			//C6-0x366
			16#366:           //接收C6送来的数据
				//Pre :=BYTE_TO_WORD(frame.data[1]) OR SHL(BYTE_TO_WORD(frame.data[2]),8);
	 			//psYyz^.Status.pressureV8:= 	(Pre-4000)/16000.0*400;	
				//Pre :=BYTE_TO_WORD(frame.data[3]) OR SHL(BYTE_TO_WORD(frame.data[4]),8);
	 			//psYyz^.Status.pressureV9:= 	(Pre-4000)/16000.0*400;	
				pos	:=BYTE_TO_WORD(frame.data[5]) OR SHL(BYTE_TO_WORD(frame.data[6]),8);
				psPVTi^.arrAddtion[1].sPlateStatus.sSensor.Current:=pos*0.1;
				pos	:=BYTE_TO_WORD(frame.data[7]) OR SHL(BYTE_TO_WORD(frame.data[8]),8);
				psPVTi^.arrAddtion[2].sPlateStatus.sSensor.Current:=pos*0.1;
				
		END_CASE
	END_FOR
	gCan.C6RxCounter := gCan.C6RxMsg.RxCounter ;
END_IF

END_FUNCTION

// Device/Application/can/swmc_C12_Rx
FUNCTION swmc_C12_Rx : BOOL
VAR_INPUT
	CNT				: UINT;
	psPVTi			: POINTER TO propValveModule_Ti;
END_VAR
VAR
	frame	 	    : Can_baseframe;
	COB_ID			: UINT;
	I				: UINT;
	Pre				: UINT;
	pos				: WORD;
END_VAR

IF gCan.C12RxMsg.RxCounter <>  gCan.C12RxCounter THEN    //接收到新的数据

	FOR  I := 1 TO  gCan.C12RxMsg.NoOfRxMessages DO
		frame :=CAN_Read_Data_SWMC(12,I);
		COB_ID :=	frame.id;    //获取ID
		CASE COB_ID OF     //根据ID解析协议
		
		
			//C12-0x3C0
			16#3C0:           //接收C12送来的数据
				pos := BYTE_TO_WORD(frame.data[ 1 ]) OR SHL(BYTE_TO_WORD(frame.data[ 2 ]),8);  	
				psPVTi^.arrPV[ 6 ].sNum[ 7 ].posVal.Current:= pos*0.1;	
				pos := BYTE_TO_WORD(frame.data[ 3 ]) OR SHL(BYTE_TO_WORD(frame.data[ 4 ]),8);  
				psPVTi^.arrPV[ 6 ].sNum[ 8 ].posVal.Current:= pos*0.1;		
				pos := BYTE_TO_WORD(frame.data[ 5 ]) OR SHL(BYTE_TO_WORD(frame.data[ 6 ]),8);  
				psPVTi^.arrPV[ 7 ].sNum[ 20 ].posVal.Current:= pos*0.1;	
				pos := BYTE_TO_WORD(frame.data[ 7 ]) OR SHL(BYTE_TO_WORD(frame.data[ 8 ]),8);  	
				psPVTi^.arrPV[ 7 ].sNum[ 21 ].posVal.Current:= pos*0.1;

			//C6-0x3C1
			16#3C1:           //接收C12送来的数据
				pos := BYTE_TO_WORD(frame.data[ 1 ]) OR SHL(BYTE_TO_WORD(frame.data[ 2 ]),8);  	
				psPVTi^.arrPV[ 7 ].sNum[ 1 ].posVal.Current:= pos*0.1;	
				pos := BYTE_TO_WORD(frame.data[ 3 ]) OR SHL(BYTE_TO_WORD(frame.data[ 4 ]),8);  	
				psPVTi^.arrPV[ 7 ].sNum[ 2 ].posVal.Current:= pos*0.1;	
				pos := BYTE_TO_WORD(frame.data[ 5 ]) OR SHL(BYTE_TO_WORD(frame.data[ 6 ]),8);  	
				psPVTi^.arrPV[ 7 ].sNum[ 3 ].posVal.Current:= pos*0.1;	
				pos := BYTE_TO_WORD(frame.data[ 7 ]) OR SHL(BYTE_TO_WORD(frame.data[ 8 ]),8);  	
				psPVTi^.arrPV[ 7 ].sNum[ 4 ].posVal.Current:= pos*0.1;
			//C6-0x3C2
			16#3C2:           //接收C12送来的数据
				pos := BYTE_TO_WORD(frame.data[ 1 ]) OR SHL(BYTE_TO_WORD(frame.data[ 2 ]),8);  	
				psPVTi^.arrPV[ 7 ].sNum[ 5 ].posVal.Current:= pos*0.1;	
				pos := BYTE_TO_WORD(frame.data[ 3 ]) OR SHL(BYTE_TO_WORD(frame.data[ 4 ]),8);  	
				psPVTi^.arrPV[ 7 ].sNum[ 6 ].posVal.Current:= pos*0.1;		
				pos := BYTE_TO_WORD(frame.data[ 5 ]) OR SHL(BYTE_TO_WORD(frame.data[ 6 ]),8);  	
				psPVTi^.arrPV[ 7 ].sNum[ 7 ].posVal.Current:= pos*0.1;		
				pos := BYTE_TO_WORD(frame.data[ 7 ]) OR SHL(BYTE_TO_WORD(frame.data[ 8 ]),8);  	
				psPVTi^.arrPV[ 7 ].sNum[ 8 ].posVal.Current:= pos*0.1;	
			//C6-0x3C3
			16#3C3:           //接收C12送来的数据
				pos := BYTE_TO_WORD(frame.data[ 1 ]) OR SHL(BYTE_TO_WORD(frame.data[ 2 ]),8);  	
				psPVTi^.arrPV[ 7 ].sNum[ 9 ].posVal.Current:= pos*0.1;		
				pos := BYTE_TO_WORD(frame.data[ 3 ]) OR SHL(BYTE_TO_WORD(frame.data[ 4 ]),8);  	
				psPVTi^.arrPV[ 7 ].sNum[ 22 ].posVal.Current:= pos*0.1;		
				pos := BYTE_TO_WORD(frame.data[ 5 ]) OR SHL(BYTE_TO_WORD(frame.data[ 6 ]),8);  	
				psPVTi^.arrPV[7 ].sNum[ 23 ].posVal.Current:= pos*0.1;		
				pos := BYTE_TO_WORD(frame.data[ 7 ]) OR SHL(BYTE_TO_WORD(frame.data[ 8 ]),8);  	
				psPVTi^.arrPV[ 1 ].sNum[ 1 ].posVal.Current:= pos*0.1;	
			//C6-0x3C4
			16#3C4:           //接收C12送来的数据
				pos := BYTE_TO_WORD(frame.data[ 1 ]) OR SHL(BYTE_TO_WORD(frame.data[ 2 ]),8);  	
				psPVTi^.arrPV[ 1 ].sNum[ 2 ].posVal.Current:= pos*0.1;		
				pos := BYTE_TO_WORD(frame.data[ 3 ]) OR SHL(BYTE_TO_WORD(frame.data[ 4 ]),8);  	
				psPVTi^.arrPV[ 7 ].sNum[ 10 ].posVal.Current:= pos*0.1;		
				pos := BYTE_TO_WORD(frame.data[ 5 ]) OR SHL(BYTE_TO_WORD(frame.data[ 6 ]),8);  	
				psPVTi^.arrPV[ 7 ].sNum[ 11 ].posVal.Current:= pos*0.1;		
				pos := BYTE_TO_WORD(frame.data[ 7 ]) OR SHL(BYTE_TO_WORD(frame.data[ 8 ]),8);  	
				psPVTi^.arrPV[7 ].sNum[ 12 ].posVal.Current:= pos*0.1;	
			//C6-0x3C5
			16#3C5:           //接收C12送来的数据
				pos := BYTE_TO_WORD(frame.data[ 1 ]) OR SHL(BYTE_TO_WORD(frame.data[ 2 ]),8);  	
				psPVTi^.arrPV[ 7 ].sNum[ 13 ].posVal.Current:= pos*0.1;		
				pos := BYTE_TO_WORD(frame.data[ 3 ]) OR SHL(BYTE_TO_WORD(frame.data[ 4 ]),8);  	
				psPVTi^.arrPV[ 7 ].sNum[ 14 ].posVal.Current:= pos*0.1;		
				pos := BYTE_TO_WORD(frame.data[ 5 ]) OR SHL(BYTE_TO_WORD(frame.data[ 6 ]),8);  	
				psPVTi^.arrPV[ 7 ].sNum[ 15 ].posVal.Current:= pos*0.1;		
				pos := BYTE_TO_WORD(frame.data[ 7 ]) OR SHL(BYTE_TO_WORD(frame.data[ 8 ]),8);  	
				psPVTi^.arrPV[ 7 ].sNum[ 16 ].posVal.Current:= pos*0.1;
			//C6-0x3C6
			16#3C6:           //接收C12送来的数据
				pos := BYTE_TO_WORD(frame.data[ 1 ]) OR SHL(BYTE_TO_WORD(frame.data[ 2 ]),8);  	
				psPVTi^.arrPV[ 7 ].sNum[ 17 ].posVal.Current:= pos*0.1;		
				pos := BYTE_TO_WORD(frame.data[ 3 ]) OR SHL(BYTE_TO_WORD(frame.data[ 4 ]),8);  	
				psPVTi^.arrPV[ 7 ].sNum[ 18 ].posVal.Current:= pos*0.1;		
				pos := BYTE_TO_WORD(frame.data[ 5 ]) OR SHL(BYTE_TO_WORD(frame.data[ 6 ]),8);  	
				psPVTi^.arrPV[ 7 ].sNum[ 19 ].posVal.Current:= pos*0.1;		
						
		
			
		END_CASE
	END_FOR
	gCan.C12RxCounter := gCan.C12RxMsg.RxCounter ;
END_IF

END_FUNCTION

// Device/Application/dataUpload/fileSaver
PROGRAM fileSaver
VAR
	path 			:STRING:='D:/log';
	intervalMs		:INT := 10;		//间隔时间
	
	init			:BOOL:= TRUE;
	i0				:INT;
	i1				:INT;	
	cCtrl			:INT;

	sav				:ARRAY[1..7,1..24] OF fileSave;
	getCtrl			:findMasterCtrl;
	getStat			:getStateByIdx;
	speed			:INT;
	nowCmd			:ARRAY[1..7,1..24] OF BOOL;
	canWrite		:ARRAY[1..7,1..24] OF BOOL;
	nowPosition		:ARRAY[1..7,1..24] OF INT;
	lastPosition	:ARRAY[1..7,1..24] OF INT;
	state			:ARRAY[1..7,1..24] OF INT;
	flag			:ARRAY[1..7,1..24] OF INT;
END_VAR
VAR CONSTANT
	aOil	:ARRAY [1..7] OF INT :=[9,11,8,8,8,8,23];		
END_VAR


//initialize
IF init THEN
	init := FALSE;
	FOR i0:=1 TO 7 DO	
	FOR i1:=1 TO aOil[i0] DO	
		sav[i0,i1](filePath := path, intervalt := intervalMs);
		sav[i0,i1].createDir(gUI.TiG_NameInit.strName[i0,i1]);
	END_FOR	
	END_FOR	
END_IF

//detect and record
FOR i0:=1 TO 7 DO		
	FOR i1:=1 TO aOil[i0] DO
		//get command
		getCtrl(grp := i0, num := i1, ctrl => cCtrl);
		nowCmd[i0,i1] := gUI.TiG.arrPV[i0].sColumn[cCtrl].bExtend OR gUI.TiG.arrPV[i0].sColumn[cCtrl].bRetract;
		//device is running
		IF nowCmd[i0 ,i1] THEN
			IF flag[i0,i1] = 0 THEN
				sav[i0,i1].new(devName :=gUI.TiG_NameInit.strName[i0,i1]);
				flag[i0,i1] := 1;
			END_IF
			//prepare data
			getData();
			//write
			sav[i0,i1].write(positionInt:=nowPosition[i0,i1],speedInt:= speed,
				stateInt := state[i0,i1]);
			
		ELSE
			//stop recording when command ends
			IF flag[i0,i1] = 1 THEN
				sav[i0,i1].write(positionInt:=nowPosition[i0,i1],speedInt:= speed,
								stateInt := state[i0,i1]);
				sav[i0,i1].close();
				flag[i0,i1] := 0;
			END_IF
		END_IF
	END_FOR	
END_FOR

ACTION getData:

//进制转换 到0.01mm
lastPosition[i0, i1] := nowPosition[i0, i1];
nowPosition[i0, i1] := REAL_TO_INT(10 * gImple.PV_GroupTi.arrPV[i0].sNum[i1].posVal.Current);

//speed  -  mm/s
IF nowPosition[i0, i1] > lastPosition[i0, i1] THEN
	speed := (nowPosition[i0, i1] - lastPosition[i0, i1]) * 100 / intervalMs;
ELSE
	speed := (lastPosition[i0, i1] - nowPosition[i0, i1]) * 100 / intervalMs;
END_IF

getStat(grp := i0, ctrl := cCtrl,state => state[i0, i1]);
END_ACTION

END_PROGRAM

// Device/Application/dataUpload/fileSave
FUNCTION_BLOCK fileSave
VAR_INPUT
	filePath 	:STRING;
	intervalt	:INT;
END_VAR
VAR_OUTPUT
END_VAR
VAR
	
	lineCount	: INT;
	fileHandle  : DWORD;
	fileName	: STRING;
END_VAR

METHOD new

	
VAR_INPUT
	devName		: STRING ;

END_VAR
VAR
	
	fileHandle0 : DWORD;
	datetime	: DATE_AND_TIME;
	UdIntms 	: UDINT;
	UdMsOffset  : UDINT;
	DTimer_Str  : STRING;
	uiYear 		: UINT; 
    uiMonth 	: UINT; 
    uiDay 		: UINT; 
    uiHour 		: UINT; 
    uiMinute 	: UINT; 
    uiSecond 	: UINT;	
	uiMsSecond	: UINT;



	 S_Time64		:  SysTime64;
	 STT			:  CurTimeEx;
	 S_Time			:  SystemTimeDate;
	 Time_Str		:  STRING;
	F_err		: DWORD;
	F_HANDL		: DWORD;

END_VAR

	STT(SystemTime:= S_Time64, TimeDate:= S_Time);
	Time_Str :='';
	Time_Str := concat(Time_Str,UINT_TO_STRING(S_Time.Year));
	Time_Str := concat(Time_Str,'-');
	Time_Str := concat(Time_Str,UINT_TO_STRING(S_Time.Month));
	Time_Str := concat(Time_Str,'-');
	Time_Str := concat(Time_Str,UINT_TO_STRING(S_Time.Day));
	Time_Str := concat(Time_Str,'_');
	Time_Str := concat(Time_Str,UINT_TO_STRING(S_Time.Hour));
	Time_Str := concat(Time_Str,'-');
	Time_Str := concat(Time_Str,UINT_TO_STRING(S_Time.Minute));
	Time_Str := concat(Time_Str,'-');
	Time_Str := concat(Time_Str,UINT_TO_STRING(S_Time.Second));
	Time_Str := concat(Time_Str,'_');
	Time_Str := concat(Time_Str,UINT_TO_STRING(S_Time.Milliseconds));

	fileName := FilePath;
	fileName := concat(fileName,'/');
	fileName := concat(fileName,devName);

	
	fileName := concat(fileName,'/');
	fileName := concat(fileName,devName);
	fileName := concat(fileName,'-');
	fileName := concat(fileName,Time_Str);
    fileName := concat(fileName,'.txt');

	fileHandle := SysFileOpen(szFile:= fileName, am:=ACCESS_MODE.AM_WRITE, pResult:= ADR(F_err));
	lineCount := -1;
	//fileHandle := SysFileOpen(szFile:= fileName, am:=ACCESS_MODE.AM_APPEND, pResult:= ADR(F_err));
END_METHOD

METHOD close
VAR_INPUT
END_VAR
IF fileHandle <> 0 THEN
	SysFileClose(hFile := fileHandle);
	fileHandle := 0;
END_IF
END_METHOD

METHOD write
VAR_INPUT

	positionInt 	:INT;
	speedInt 		:INT;
	stateInt		:INT;
	
END_VAR
VAR
	data		: STRING;
	F_err		: DWORD;
	tempInt		: INT;
END_VAR

IF fileHandle <> 0 THEN
	lineCount := lineCount + 1;
	tempInt	:= lineCount * intervalt;
	data := INT_TO_STRING(lineCount);
	data := concat(data,'$T$T');
	data := concat(data, INT_TO_STRING(tempInt));
	IF tempInt < 1000 THEN
		data := concat(data,'$T');
	END_IF
	data := concat(data,'$T$T');
	data := concat(data,INT_TO_STRING(positionInt));
	data := concat(data,'$T');
	data := concat(data,INT_TO_STRING(speedInt));
	data := concat(data,'$T');
	data := concat(data,INT_TO_STRING(stateInt));
	data := concat(data,'$R');
	
	SysFileWrite(hFile:=fileHandle , pbyBuffer:= ADR(data) , ulSize:= SysStrLen(data) , pResult:= ADR(F_err));		// 写入数据

END_IF
END_METHOD

METHOD createDir
VAR_INPUT
	devName		: STRING ;
END_VAR
VAR
	filePath1	:STRING;
END_VAR
filePath1 := FilePath;
filePath1 := concat(filePath1,'/');
filePath1 := concat(filePath1,devName);
SysDirCreate2(filePath1, TRUE);
END_METHOD

END_FUNCTION_BLOCK

// Device/Application/public_datum/datarecord/datSave
FUNCTION_BLOCK datSave
VAR_INPUT
	Data_Arry	: ARRAY[1..200] OF UINT;	// 数据输入 一次最大可以写入200个数据
	Num			: UINT;						// 存储数据个数
	FilePath 	: STRING := 'C:/DataSave'; 	// 存储文件夹
	cycle		: TIME;						// 更新一个文件夹时间
END_VAR
VAR_OUTPUT
END_VAR
VAR
	datetime	: DATE_AND_TIME;
	uiYear 		: UINT; 
    uiMonth 	: UINT; 
    uiDay 		: UINT; 
    uiHour 		: UINT; 
    uiMinute 	: UINT; 
    uiSecond 	: UINT;	
	uiMsSecond	: UINT;
	Last_S		: UINT:=100;
	UdMsOffset  : UDINT;
	UdIntms 	: UDINT;
	DTimer_Arry : ARRAY[1..7] OF UINT;
END_VAR
VAR
	File_Init	: BOOL :=TRUE;
	Frame_Cnt	: LINT;
	Data_Save_Init :BOOL:=TRUE;
	New_File_Ton: TON;
	Filename	: STRING;
	F_HANDL		: DWORD;
	F_err		: DWORD;
	F_pos		: DWORD;
END_VAR

datetime:=GetDateTime();   //获取时间
DTU.DTSplit(
		dtDateAndTime:= datetime, 
		puiYear:= ADR(uiYear), 
		puiMonth:=  ADR(uiMonth), 
		puiDay:=  ADR(uiDay), 
		puiHour:=  ADR(uiHour), 
		puiMinute:=  ADR(uiMinute), 
		puiSecond:= ADR(uiSecond) );

IF  Data_Save_Init THEN			//数据存储初始化
	IF uiSecond = Last_S +1 OR  uiSecond = Last_S -59 THEN
		UdMsOffset := SysTimeGetMs();
		Last_S :=  uiSecond;
	ELSE
		Last_S :=  uiSecond;
		RETURN;
	END_IF
    Data_Save_Init := FALSE;
END_IF

IF 	File_Init  THEN          //创建文件
	Filename := FilePath;
	Filename := concat(Filename,'/');
	Filename := concat(Filename,UINT_TO_STRING(uiYear));
	Filename := concat(Filename,'_');
	Filename := concat(Filename,UINT_TO_STRING(uiMonth));
	Filename := concat(Filename,'_');
	Filename := concat(Filename,UINT_TO_STRING(uiDay));
	Filename := concat(Filename,'_');
	Filename := concat(Filename,UINT_TO_STRING(uiHour+8));
 	Filename := concat(Filename,'_');
	Filename := concat(Filename,UINT_TO_STRING(uiMinute));
	Filename := concat(Filename,'_');
	Filename := concat(Filename,UINT_TO_STRING(uiSecond));
    Filename := concat(Filename,'_Data.bin');
	Frame_Cnt := 0;
	F_HANDL :=SysFileOpen(szFile:= Filename, am:=ACCESS_MODE.AM_WRITE, pResult:= ADR(F_err));  //创建新文件
	SysFileClose(hFile:=F_HANDL );
	File_Init := FALSE;
	New_File_Ton(IN:= FALSE , PT:= cycle, Q=> , ET=> );  //复位
END_IF

New_File_Ton(IN:= TRUE , PT:= cycle, Q=> , ET=> );			//4小时创建一个新文件
IF New_File_Ton.Q THEN
	File_Init := TRUE;	
END_IF



UdIntms := SysTimeGetMs();
DTimer_Arry[1] := uiYear;
DTimer_Arry[2] := uiMonth;
DTimer_Arry[3] := uiDay;
DTimer_Arry[4] := uiHour+8;
DTimer_Arry[5] := uiMinute;
DTimer_Arry[6] := uiSecond;
DTimer_Arry[7] := UDINT_TO_UINT((UdIntms - UdMsOffset)MOD 1000);

Frame_Cnt := Frame_Cnt + 1;    	//帧计数增加

F_HANDL :=SysFileOpen(szFile:= Filename, am:=ACCESS_MODE.AM_APPEND, pResult:= ADR(F_err));  //打开文件
SysFileGetPos(hFile:= F_HANDL , pulPos:= ADR(F_pos));		//获取文件位置
SysFileSetPos(hFile:= F_HANDL, ulOffset:= 0);	//设置帧位置
SysFileWrite(hFile:=F_HANDL , pbyBuffer:= ADR(Frame_Cnt) , ulSize:= SIZEOF(Frame_Cnt) , pResult:= ADR(F_err));    //修改总帧数
IF F_pos <> 0 THEN		//不是新文件，设置写入位置
	SysFileSetPos(hFile:= F_HANDL, ulOffset:= F_pos);
END_IF
SysFileWrite(hFile:=F_HANDL , pbyBuffer:= ADR(DTimer_Arry) , ulSize:= SIZEOF(DTimer_Arry) , pResult:= ADR(F_err));  // 保存时间
SysFileWrite(hFile:=F_HANDL , pbyBuffer:= ADR(Data_Arry) , ulSize:= SIZEOF(UINT)*Num , pResult:= ADR(F_err));		// 保存数据
SysFileClose(hFile:=F_HANDL );

END_FUNCTION_BLOCK

// Device/Application/rail_ceiling/positionRecord
PROGRAM positionRecord
VAR
	arrPosVal			:ARRAY[1..200] OF UINT;
	fbDatSav			:DatSave;
	iT1					:UINT;
	iT2					:UINT;
	iNum				:UINT;
END_VAR
VAR CONSTANT
	aOil	:ARRAY [1..7] OF UINT :=[9,11,8,8,8,8,23];		
END_VAR

iNum:=1;
FOR iT1:=1 TO 7 DO
	FOR iT2:=1 TO aOil[iT1] DO
		arrPosVal[iNum]:=REAL_TO_UINT(gImple.PV_GroupTi.arrPV[iT1].sNum[iT2].posVal.Current);
		iNum:=iNum+1;
	END_FOR
END_FOR
fbDatSav(Data_Arry:=arrPosVal , Num:= 75 , FilePath:= 'D:/DataSave', cycle:= T#7200S);

END_PROGRAM

// Device/Application/public_datum/cmdcheck/syncUnitCheck
FUNCTION_BLOCK syncUnitCheck
VAR_INPUT
	arrPosVal	:ARRAY  [1..2] OF OilBlockUnit_Status_PosVal;

	cmdAct		:cmdStat;
	
END_VAR
VAR_OUTPUT
	bFetch		:BOOL;
END_VAR
VAR
	iCheck			:INT;
	iNum			:INT;				//有值的位移传感器值
	outStat			:ARRAY[1..2] OF OilBlockUnit_Status_Loc;
	iTemp			:INT;
	bAllDone		:BOOL;
END_VAR

iNum:=0;
FOR iTemp :=1 TO 2 DO
	IF arrPosVal[iTemp].Extend <> 0 THEN
		iNum:=iNum+1;
	END_IF
END_FOR
FOR iCheck:=1 TO iNum DO
	outStat[iCheck]	:=fGetUnitStat(arrPosVal[iCheck].Extend,arrPosVal[iCheck].Retract,arrPosVal[iCheck].Current,2.0);
END_FOR


bAllDone:=TRUE;

	//有一个未到指令位置则未完成
	CASE cmdAct OF 
		cmdStat.cExtend:
			FOR iCheck:=1 TO iNum DO
				IF outStat[iCheck]<>OilBlockUnit_Status_Loc.eExtended THEN
					bAllDone:=FALSE;
				END_IF
			END_FOR
		cmdStat.cRetract:
			FOR iCheck:=1 TO iNum DO
				IF outStat[iCheck]<>OilBlockUnit_Status_Loc.eRetracted THEN
					bAllDone:=FALSE;
				END_IF
			END_FOR	
		cmdStat.cStop:
			
	END_CASE

IF bAllDone THEN
	bFetch	:= TRUE;
ELSE
	bFetch	:= FALSE;
END_IF

END_FUNCTION_BLOCK

// Device/Application/display/Module/OilBlock_PrimButton
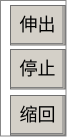
VISUALIZATION OilBlock_PrimButton  // 67x137
VAR_IN_OUT
	extendButton		: BOOL;
	retractButton		: BOOL;
	stopButton			: BOOL;
	
END_VAR
    Button (10,95 55x40), "缩回"
        toggle retractButton
    Button (10,49 55x40), "停止"
        toggle stopButton
    Button (10,5 55x40), "伸出"
        toggle extendButton
END_VISUALIZATION

// Device/Application/display/Module/OilBlock_PrimInfo
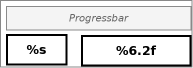
VISUALIZATION OilBlock_PrimInfo  // 193x68
VAR_IN_OUT
	nameStr		:STRING;
	posVal		:REAL;
	percentBar	:REAL;
END_VAR
    RoundedRectangle (6,34 61x31), "%s", text variable: nameStr
    RoundedRectangle (81,35 110x31), "%6.2f", text variable: posVal
    Progressbar (6,6 185x24), variable: percentBar
END_VISUALIZATION

// Device/Application/display/Module/ModuleX2
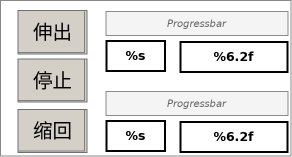
VISUALIZATION ModuleX2  // 292x157
VAR_IN_OUT
	extendButton		: BOOL;
	retractButton		: BOOL;
	stopButton			: BOOL;
	
	nameStr1			:STRING;
	posVal1				:REAL;
	percentBar1			:REAL;
	nameStr2			:STRING;
	posVal2				:REAL;
	percentBar2			:REAL;
END_VAR
    Group (5,5 285x150)
        Frame (0,0 85x150)
            shows OilBlock_PrimButton(extendButton := extendButton, retractButton := retractButton, stopButton := stopButton)
        Frame (95,0 190x70)
            shows OilBlock_PrimInfo(nameStr := nameStr1, posVal := posVal1, percentBar := percentBar1)
        Frame (95,80 190x70)
            shows OilBlock_PrimInfo(nameStr := nameStr2, posVal := posVal2, percentBar := percentBar2)
END_VISUALIZATION

// Device/Application/display/Module/ModuleX1
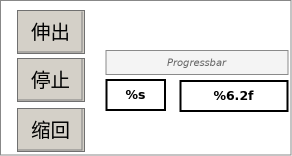
VISUALIZATION ModuleX1  // 292x156
VAR_IN_OUT
	extendButton		: BOOL;
	retractButton		: BOOL;
	stopButton			: BOOL;
	
	nameStr				:STRING;
	posVal				:REAL;
	percentBar			:REAL;
END_VAR
    Group (5,5 285x149)
        Frame (0,0 82x149)
            shows OilBlock_PrimButton(extendButton := extendButton, retractButton := retractButton, stopButton := stopButton)
        Frame (95,39 190x70)
            shows OilBlock_PrimInfo(nameStr := nameStr, posVal := posVal, percentBar := percentBar)
END_VISUALIZATION

// Device/Application/display/Module/ModuleX3
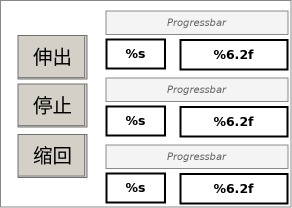
VISUALIZATION ModuleX3  // 292x208
VAR_IN_OUT
	extendButton		: BOOL;
	retractButton		: BOOL;
	stopButton			: BOOL;
	
	nameStr1			:STRING;
	posVal1				:REAL;
	percentBar1			:REAL;
	nameStr2			:STRING;
	posVal2				:REAL;
	percentBar2			:REAL;
	nameStr3			:STRING;
	posVal3				:REAL;
	percentBar3			:REAL;
END_VAR
    Group (5,5 285x201)
        Frame (0,25 85x150)
            shows OilBlock_PrimButton(extendButton := extendButton, retractButton := retractButton, stopButton := stopButton)
        Frame (95,0 190x67)
            shows OilBlock_PrimInfo(nameStr := nameStr1, posVal := posVal1, percentBar := percentBar1)
        Frame (95,67 190x67)
            shows OilBlock_PrimInfo(nameStr := nameStr2, posVal := posVal2, percentBar := percentBar2)
        Frame (95,134 190x67)
            shows OilBlock_PrimInfo(nameStr := nameStr3, posVal := posVal3, percentBar := percentBar3)
END_VISUALIZATION

// Device/Application/display/Module/ModuleX8
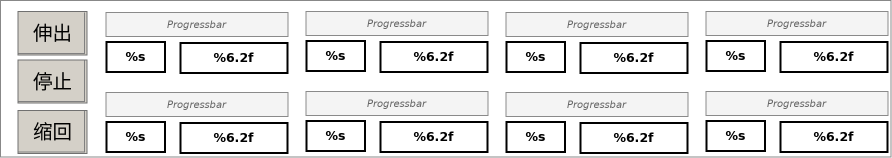
VISUALIZATION ModuleX8  // 892x158
VAR_IN_OUT
	extendButton		: BOOL;
	retractButton		: BOOL;
	stopButton			: BOOL;
	
	nameStr1			:STRING;
	posVal1				:REAL;
	percentBar1			:REAL;
	
	nameStr2			:STRING;
	posVal2				:REAL;
	percentBar2			:REAL;
	
	nameStr3			:STRING;
	posVal3				:REAL;
	percentBar3			:REAL;
	
	nameStr4			:STRING;
	posVal4				:REAL;
	percentBar4			:REAL;
	
	nameStr5			:STRING;
	posVal5				:REAL;
	percentBar5			:REAL;
	
	nameStr6			:STRING;
	posVal6				:REAL;
	percentBar6			:REAL;
	
	nameStr7			:STRING;
	posVal7				:REAL;
	percentBar7			:REAL;
	
	nameStr8			:STRING;
	posVal8				:REAL;
	percentBar8			:REAL;	
	
END_VAR
    Group (5,5 885x151)
        Frame (0,1 85x150)
            shows OilBlock_PrimButton(extendButton := extendButton, retractButton := retractButton, stopButton := stopButton)
        Group (95,0 390x151)
            Group (0,1 190x150)
                Frame (0,0 190x70)
                    shows OilBlock_PrimInfo(nameStr := nameStr1, posVal := posVal1, percentBar := percentBar1)
                Frame (0,80 190x70)
                    shows OilBlock_PrimInfo(nameStr := nameStr2, posVal := posVal2, percentBar := percentBar2)
            Frame (200,0 190x70)
                shows OilBlock_PrimInfo(nameStr := nameStr3, posVal := posVal3, percentBar := percentBar3)
            Frame (200,80 190x70)
                shows OilBlock_PrimInfo(nameStr := nameStr4, posVal := posVal4, percentBar := percentBar4)
        Frame (495,1 190x70)
            shows OilBlock_PrimInfo(nameStr := nameStr5, posVal := posVal5, percentBar := percentBar5)
        Frame (495,81 190x70)
            shows OilBlock_PrimInfo(nameStr := nameStr6, posVal := posVal6, percentBar := percentBar6)
        Frame (695,0 190x70)
            shows OilBlock_PrimInfo(nameStr := nameStr7, posVal := posVal7, percentBar := percentBar7)
        Frame (695,80 190x70)
            shows OilBlock_PrimInfo(nameStr := nameStr8, posVal := posVal8, percentBar := percentBar8)
END_VISUALIZATION

// Device/Application/display/Module/ModuleX4
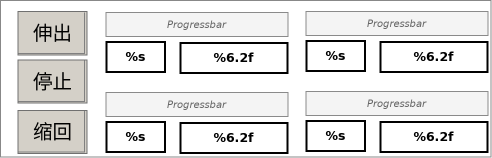
VISUALIZATION ModuleX4  // 492x158
VAR_IN_OUT
	extendButton		: BOOL;
	retractButton		: BOOL;
	stopButton			: BOOL;
	
	nameStr1			:STRING;
	posVal1				:REAL;
	percentBar1			:REAL;
	nameStr2			:STRING;
	posVal2				:REAL;
	percentBar2			:REAL;
	nameStr3			:STRING;
	posVal3				:REAL;
	percentBar3			:REAL;
	nameStr4			:STRING;
	posVal4				:REAL;
	percentBar4			:REAL;
	
	
END_VAR
    Group (5,5 485x151)
        Frame (0,1 85x150)
            shows OilBlock_PrimButton(extendButton := extendButton, retractButton := retractButton, stopButton := stopButton)
        Group (95,1 190x150)
            Frame (0,0 190x70)
                shows OilBlock_PrimInfo(nameStr := nameStr1, posVal := posVal1, percentBar := percentBar1)
            Frame (0,80 190x70)
                shows OilBlock_PrimInfo(nameStr := nameStr2, posVal := posVal2, percentBar := percentBar2)
        Frame (295,0 190x70)
            shows OilBlock_PrimInfo(nameStr := nameStr3, posVal := posVal3, percentBar := percentBar3)
        Frame (295,80 190x70)
            shows OilBlock_PrimInfo(nameStr := nameStr4, posVal := posVal4, percentBar := percentBar4)
END_VISUALIZATION

// Device/Application/display/Module/ModuleX5
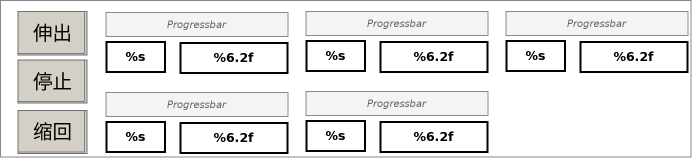
VISUALIZATION ModuleX5  // 692x158
VAR_IN_OUT
	extendButton		: BOOL;
	retractButton		: BOOL;
	stopButton			: BOOL;
	
	nameStr1			:STRING;
	posVal1				:REAL;
	percentBar1			:REAL;
	nameStr2			:STRING;
	posVal2				:REAL;
	percentBar2			:REAL;
	nameStr3			:STRING;
	posVal3				:REAL;
	percentBar3			:REAL;
	nameStr4			:STRING;
	posVal4				:REAL;
	percentBar4			:REAL;
	nameStr5			:STRING;
	posVal5				:REAL;
	percentBar5			:REAL;
	
	
END_VAR
    Group (5,5 685x151)
        Frame (0,1 85x150)
            shows OilBlock_PrimButton(extendButton := extendButton, retractButton := retractButton, stopButton := stopButton)
        Group (95,1 190x150)
            Frame (0,0 190x70)
                shows OilBlock_PrimInfo(nameStr := nameStr1, posVal := posVal1, percentBar := percentBar1)
            Frame (0,80 190x70)
                shows OilBlock_PrimInfo(nameStr := nameStr2, posVal := posVal2, percentBar := percentBar2)
        Frame (295,0 190x70)
            shows OilBlock_PrimInfo(nameStr := nameStr3, posVal := posVal3, percentBar := percentBar3)
        Frame (295,80 190x70)
            shows OilBlock_PrimInfo(nameStr := nameStr4, posVal := posVal4, percentBar := percentBar4)
        Frame (495,0 190x70)
            shows OilBlock_PrimInfo(nameStr := nameStr5, posVal := posVal5, percentBar := percentBar5)
END_VISUALIZATION

// Device/Application/display/OrigTi/Ceiling_Rail2
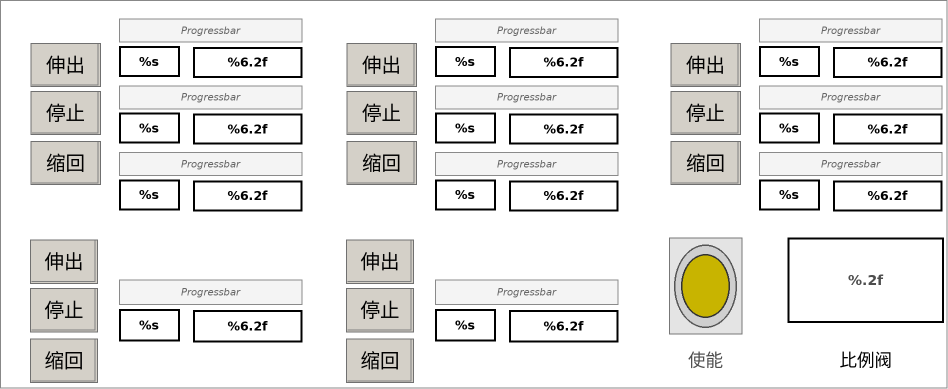
VISUALIZATION Ceiling_Rail2  // 948x389
    Frame (13,8 293x207)
        shows ModuleX3(extendButton := gUI.TiG.arrPV[2].sColumn[1].bExtend, retractButton := gUI.TiG.arrPV[2].sColumn[1].bRetract, stopButton := gUI.TiG.arrPV[2].sColumn[1].bStop, nameStr1 := gUI.TiG.arrPV[2].sNum[1].strName, posVal1 := gUI.TiG.arrPV[2].sNum[1].rPosition, percentBar1 := gUI.TiG.arrPV[2].sNum[1].rPercent, nameStr2 := gUI.TiG.arrPV[2].sNum[2].strName, posVal2 := gUI.TiG.arrPV[2].sNum[2].rPosition, percentBar2 := gUI.TiG.arrPV[2].sNum[2].rPercent, nameStr3 := gUI.TiG.arrPV[2].sNum[3].strName, posVal3 := gUI.TiG.arrPV[2].sNum[3].rPosition, percentBar3 := gUI.TiG.arrPV[2].sNum[3].rPercent)
    Frame (13,229 293x158)
        shows ModuleX1(extendButton := gUI.TiG.arrPV[2].sColumn[2].bExtend, retractButton := gUI.TiG.arrPV[2].sColumn[2].bRetract, stopButton := gUI.TiG.arrPV[2].sColumn[2].bStop, nameStr := gUI.TiG.arrPV[2].sNum[4].strName, posVal := gUI.TiG.arrPV[2].sNum[4].rPosition, percentBar := gUI.TiG.arrPV[2].sNum[4].rPercent)
    Frame (329,8 293x207)
        shows ModuleX3(extendButton := gUI.TiG.arrPV[2].sColumn[3].bExtend, retractButton := gUI.TiG.arrPV[2].sColumn[3].bRetract, stopButton := gUI.TiG.arrPV[2].sColumn[3].bStop, nameStr1 := gUI.TiG.arrPV[2].sNum[5].strName, posVal1 := gUI.TiG.arrPV[2].sNum[5].rPosition, percentBar1 := gUI.TiG.arrPV[2].sNum[5].rPercent, nameStr2 := gUI.TiG.arrPV[2].sNum[6].strName, posVal2 := gUI.TiG.arrPV[2].sNum[6].rPosition, percentBar2 := gUI.TiG.arrPV[2].sNum[6].rPercent, nameStr3 := gUI.TiG.arrPV[2].sNum[7].strName, posVal3 := gUI.TiG.arrPV[2].sNum[7].rPosition, percentBar3 := gUI.TiG.arrPV[2].sNum[7].rPercent)
    Frame (329,229 293x158)
        shows ModuleX1(extendButton := gUI.TiG.arrPV[2].sColumn[4].bExtend, retractButton := gUI.TiG.arrPV[2].sColumn[4].bRetract, stopButton := gUI.TiG.arrPV[2].sColumn[4].bStop, nameStr := gUI.TiG.arrPV[2].sNum[8].strName, posVal := gUI.TiG.arrPV[2].sNum[8].rPosition, percentBar := gUI.TiG.arrPV[2].sNum[8].rPercent)
    Frame (653,8 293x207)
        shows ModuleX3(extendButton := gUI.TiG.arrPV[2].sColumn[5].bExtend, retractButton := gUI.TiG.arrPV[2].sColumn[5].bRetract, stopButton := gUI.TiG.arrPV[2].sColumn[5].bStop, nameStr1 := gUI.TiG.arrPV[2].sNum[9].strName, posVal1 := gUI.TiG.arrPV[2].sNum[9].rPosition, percentBar1 := gUI.TiG.arrPV[2].sNum[9].rPercent, nameStr2 := gUI.TiG.arrPV[2].sNum[10].strName, posVal2 := gUI.TiG.arrPV[2].sNum[10].rPosition, percentBar2 := gUI.TiG.arrPV[2].sNum[10].rPercent, nameStr3 := gUI.TiG.arrPV[2].sNum[11].strName, posVal3 := gUI.TiG.arrPV[2].sNum[11].rPosition, percentBar3 := gUI.TiG.arrPV[2].sNum[11].rPercent)
    Frame (653,229 293x158)
        shows ModuleDTD(enable := gUI.TiG.arrPV[2].bPVD_enable, propPercent := gUI.TiG.arrPV[2].rPVDPercent)
END_VISUALIZATION

// Device/Application/display/Module/ModuleDTD
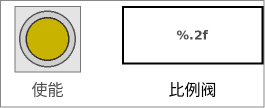
VISUALIZATION ModuleDTD  // 265x108
VAR_IN_OUT
	enable			:BOOL;
	propPercent		:REAL;
END_VAR
    Rectangle (122,6 141x58), "%.2f", text variable: propPercent
        OnMouseDown: write the text variable via Default, min 0, max 100
    Label (122,74 141x32), "比例阀"
    PushSwitchLed (13,6 69x66), variable: enable, behaviour: TOGGLE, style: Switch-PushSwitchLed-Yellow
    Label (13,74 69x32), "使能"
END_VISUALIZATION

// Device/Application/display/OrigTi/Ceiling_Rail1
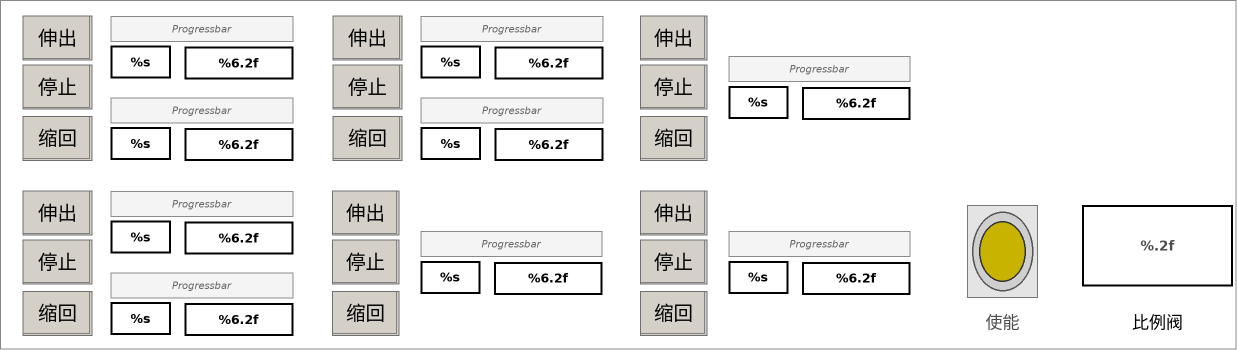
VISUALIZATION Ceiling_Rail1  // 1237x350
    Frame (5,5 292x160)
        shows ModuleX2(extendButton := gUI.TiG.arrPV[1].sColumn[1].bExtend, retractButton := gUI.TiG.arrPV[1].sColumn[1].bRetract, stopButton := gUI.TiG.arrPV[1].sColumn[1].bStop, nameStr1 := gUI.TiG.arrPV[1].sNum[1].strName, posVal1 := gUI.TiG.arrPV[1].sNum[1].rPosition, percentBar1 := gUI.TiG.arrPV[1].sNum[1].rPercent, nameStr2 := gUI.TiG.arrPV[1].sNum[2].strName, posVal2 := gUI.TiG.arrPV[1].sNum[2].rPosition, percentBar2 := gUI.TiG.arrPV[1].sNum[2].rPercent)
    Frame (315,5 292x160)
        shows ModuleX2(extendButton := gUI.TiG.arrPV[1].sColumn[2].bExtend, retractButton := gUI.TiG.arrPV[1].sColumn[2].bRetract, stopButton := gUI.TiG.arrPV[1].sColumn[2].bStop, nameStr1 := gUI.TiG.arrPV[1].sNum[3].strName, posVal1 := gUI.TiG.arrPV[1].sNum[3].rPosition, percentBar1 := gUI.TiG.arrPV[1].sNum[3].rPercent, nameStr2 := gUI.TiG.arrPV[1].sNum[4].strName, posVal2 := gUI.TiG.arrPV[1].sNum[4].rPosition, percentBar2 := gUI.TiG.arrPV[1].sNum[4].rPercent)
    Frame (5,180 292x160)
        shows ModuleX2(extendButton := gUI.TiG.arrPV[1].sColumn[4].bExtend, retractButton := gUI.TiG.arrPV[1].sColumn[4].bRetract, stopButton := gUI.TiG.arrPV[1].sColumn[4].bStop, nameStr1 := gUI.TiG.arrPV[1].sNum[6].strName, posVal1 := gUI.TiG.arrPV[1].sNum[6].rPosition, percentBar1 := gUI.TiG.arrPV[1].sNum[6].rPercent, nameStr2 := gUI.TiG.arrPV[1].sNum[7].strName, posVal2 := gUI.TiG.arrPV[1].sNum[7].rPosition, percentBar2 := gUI.TiG.arrPV[1].sNum[7].rPercent)
    Frame (952,197 283x151)
        shows ModuleDTD(enable := gUI.TiG.arrPV[1].bPVD_enable, propPercent := gUI.TiG.arrPV[1].rPVDPercent)
    Frame (623,5 291x160)
        shows ModuleX1(extendButton := gUI.TiG.arrPV[1].sColumn[3].bExtend, retractButton := gUI.TiG.arrPV[1].sColumn[3].bRetract, stopButton := gUI.TiG.arrPV[1].sColumn[3].bStop, nameStr := gUI.TiG.arrPV[1].sNum[5].strName, posVal := gUI.TiG.arrPV[1].sNum[5].rPosition, percentBar := gUI.TiG.arrPV[1].sNum[5].rPercent)
    Frame (315,180 291x160)
        shows ModuleX1(extendButton := gUI.TiG.arrPV[1].sColumn[5].bExtend, retractButton := gUI.TiG.arrPV[1].sColumn[5].bRetract, stopButton := gUI.TiG.arrPV[1].sColumn[5].bStop, nameStr := gUI.TiG.arrPV[1].sNum[8].strName, posVal := gUI.TiG.arrPV[1].sNum[8].rPosition, percentBar := gUI.TiG.arrPV[1].sNum[8].rPercent)
    Frame (623,180 291x160)
        shows ModuleX1(extendButton := gUI.TiG.arrPV[1].sColumn[6].bExtend, retractButton := gUI.TiG.arrPV[1].sColumn[6].bRetract, stopButton := gUI.TiG.arrPV[1].sColumn[6].bStop, nameStr := gUI.TiG.arrPV[1].sNum[9].strName, posVal := gUI.TiG.arrPV[1].sNum[9].rPosition, percentBar := gUI.TiG.arrPV[1].sNum[9].rPercent)
END_VISUALIZATION

// Device/Application/display/OrigTi/Ceiling_Rail_345
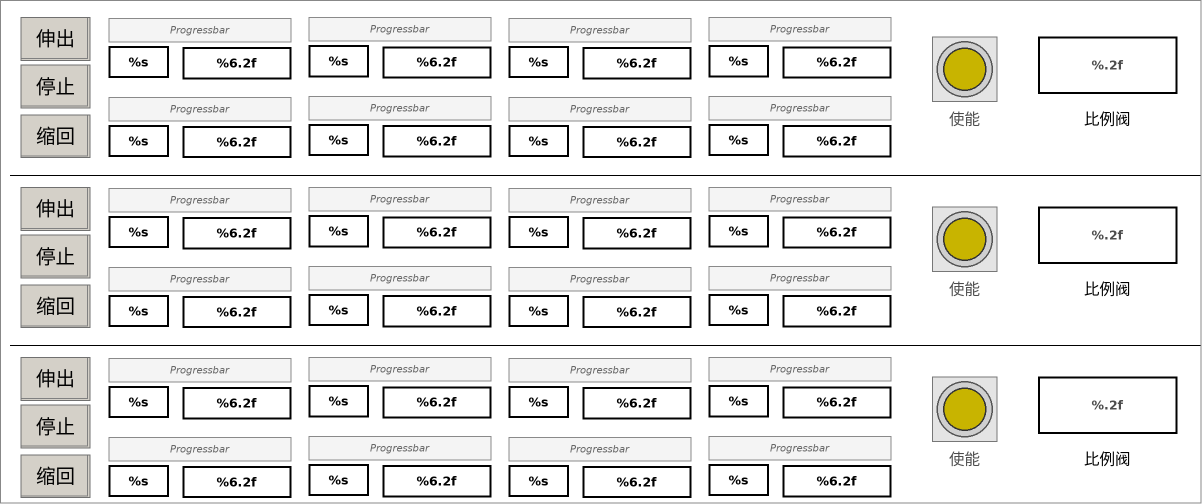
VISUALIZATION Ceiling_Rail_345  // 1202x504
    Frame (3,6 892x156)
        shows ModuleX8(extendButton := gUI.TiG.arrPV[3].sColumn[1].bExtend, retractButton := gUI.TiG.arrPV[3].sColumn[1].bRetract, stopButton := gUI.TiG.arrPV[3].sColumn[1].bStop, nameStr1 := gUI.TiG.arrPV[3].sNum[1].strName, posVal1 := gUI.TiG.arrPV[3].sNum[1].rPosition, percentBar1 := gUI.TiG.arrPV[3].sNum[1].rPercent, nameStr2 := gUI.TiG.arrPV[3].sNum[2].strName, posVal2 := gUI.TiG.arrPV[3].sNum[2].rPosition, percentBar2 := gUI.TiG.arrPV[3].sNum[2].rPercent, nameStr3 := gUI.TiG.arrPV[3].sNum[3].strName, posVal3 := gUI.TiG.arrPV[3].sNum[3].rPosition, percentBar3 := gUI.TiG.arrPV[3].sNum[3].rPercent, nameStr4 := gUI.TiG.arrPV[3].sNum[4].strName, posVal4 := gUI.TiG.arrPV[3].sNum[4].rPosition, percentBar4 := gUI.TiG.arrPV[3].sNum[4].rPercent, nameStr5 := gUI.TiG.arrPV[3].sNum[5].strName, posVal5 := gUI.TiG.arrPV[3].sNum[5].rPosition, percentBar5 := gUI.TiG.arrPV[3].sNum[5].rPercent, nameStr6 := gUI.TiG.arrPV[3].sNum[6].strName, posVal6 := gUI.TiG.arrPV[3].sNum[6].rPosition, percentBar6 := gUI.TiG.arrPV[3].sNum[6].rPercent, nameStr7 := gUI.TiG.arrPV[3].sNum[7].strName, posVal7 := gUI.TiG.arrPV[3].sNum[7].rPosition, percentBar7 := gUI.TiG.arrPV[3].sNum[7].rPercent, nameStr8 := gUI.TiG.arrPV[3].sNum[8].strName, posVal8 := gUI.TiG.arrPV[3].sNum[8].rPosition, percentBar8 := gUI.TiG.arrPV[3].sNum[8].rPercent)
    Frame (3,176 892x156)
        shows ModuleX8(extendButton := gUI.TiG.arrPV[4].sColumn[1].bExtend, retractButton := gUI.TiG.arrPV[4].sColumn[1].bRetract, stopButton := gUI.TiG.arrPV[4].sColumn[1].bStop, nameStr1 := gUI.TiG.arrPV[4].sNum[1].strName, posVal1 := gUI.TiG.arrPV[4].sNum[1].rPosition, percentBar1 := gUI.TiG.arrPV[4].sNum[1].rPercent, nameStr2 := gUI.TiG.arrPV[4].sNum[2].strName, posVal2 := gUI.TiG.arrPV[4].sNum[2].rPosition, percentBar2 := gUI.TiG.arrPV[4].sNum[2].rPercent, nameStr3 := gUI.TiG.arrPV[4].sNum[3].strName, posVal3 := gUI.TiG.arrPV[4].sNum[3].rPosition, percentBar3 := gUI.TiG.arrPV[4].sNum[3].rPercent, nameStr4 := gUI.TiG.arrPV[4].sNum[4].strName, posVal4 := gUI.TiG.arrPV[4].sNum[4].rPosition, percentBar4 := gUI.TiG.arrPV[4].sNum[4].rPercent, nameStr5 := gUI.TiG.arrPV[4].sNum[5].strName, posVal5 := gUI.TiG.arrPV[4].sNum[5].rPosition, percentBar5 := gUI.TiG.arrPV[4].sNum[5].rPercent, nameStr6 := gUI.TiG.arrPV[4].sNum[6].strName, posVal6 := gUI.TiG.arrPV[4].sNum[6].rPosition, percentBar6 := gUI.TiG.arrPV[4].sNum[6].rPercent, nameStr7 := gUI.TiG.arrPV[4].sNum[7].strName, posVal7 := gUI.TiG.arrPV[4].sNum[7].rPosition, percentBar7 := gUI.TiG.arrPV[4].sNum[7].rPercent, nameStr8 := gUI.TiG.arrPV[4].sNum[8].strName, posVal8 := gUI.TiG.arrPV[4].sNum[8].rPosition, percentBar8 := gUI.TiG.arrPV[4].sNum[8].rPercent)
    Frame (3,346 892x156)
        shows ModuleX8(extendButton := gUI.TiG.arrPV[5].sColumn[1].bExtend, retractButton := gUI.TiG.arrPV[5].sColumn[1].bRetract, stopButton := gUI.TiG.arrPV[5].sColumn[1].bStop, nameStr1 := gUI.TiG.arrPV[5].sNum[1].strName, posVal1 := gUI.TiG.arrPV[5].sNum[1].rPosition, percentBar1 := gUI.TiG.arrPV[5].sNum[1].rPercent, nameStr2 := gUI.TiG.arrPV[5].sNum[2].strName, posVal2 := gUI.TiG.arrPV[5].sNum[2].rPosition, percentBar2 := gUI.TiG.arrPV[5].sNum[2].rPercent, nameStr3 := gUI.TiG.arrPV[5].sNum[3].strName, posVal3 := gUI.TiG.arrPV[5].sNum[3].rPosition, percentBar3 := gUI.TiG.arrPV[5].sNum[3].rPercent, nameStr4 := gUI.TiG.arrPV[5].sNum[4].strName, posVal4 := gUI.TiG.arrPV[5].sNum[4].rPosition, percentBar4 := gUI.TiG.arrPV[5].sNum[4].rPercent, nameStr5 := gUI.TiG.arrPV[5].sNum[5].strName, posVal5 := gUI.TiG.arrPV[5].sNum[5].rPosition, percentBar5 := gUI.TiG.arrPV[5].sNum[5].rPercent, nameStr6 := gUI.TiG.arrPV[5].sNum[6].strName, posVal6 := gUI.TiG.arrPV[5].sNum[6].rPosition, percentBar6 := gUI.TiG.arrPV[5].sNum[6].rPercent, nameStr7 := gUI.TiG.arrPV[5].sNum[7].strName, posVal7 := gUI.TiG.arrPV[5].sNum[7].rPosition, percentBar7 := gUI.TiG.arrPV[5].sNum[7].rPercent, nameStr8 := gUI.TiG.arrPV[5].sNum[8].strName, posVal8 := gUI.TiG.arrPV[5].sNum[8].rPosition, percentBar8 := gUI.TiG.arrPV[5].sNum[8].rPercent)
    Frame (918,31 261x106)
        shows ModuleDTD(enable := gUI.TiG.arrPV[3].bPVD_enable, propPercent := gUI.TiG.arrPV[3].rPVDPercent)
    Frame (918,201 261x106)
        shows ModuleDTD(enable := gUI.TiG.arrPV[4].bPVD_enable, propPercent := gUI.TiG.arrPV[4].rPVDPercent)
    Frame (918,371 261x106)
        shows ModuleDTD(enable := gUI.TiG.arrPV[5].bPVD_enable, propPercent := gUI.TiG.arrPV[5].rPVDPercent)
    Line (10,175) (1200,175)
    Line (10,345) (1200,345)
END_VISUALIZATION

// Device/Application/display/OrigTi/Ceiling_Rail6
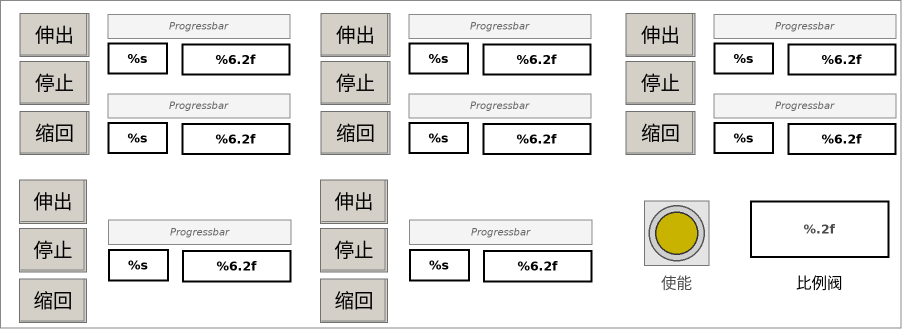
VISUALIZATION Ceiling_Rail6  // 902x329
    Frame (2,169 293x158)
        shows ModuleX1(extendButton := gUI.TiG.arrPV[6].sColumn[2].bExtend, retractButton := gUI.TiG.arrPV[6].sColumn[2].bRetract, stopButton := gUI.TiG.arrPV[6].sColumn[2].bStop, nameStr := gUI.TiG.arrPV[6].sNum[3].strName, posVal := gUI.TiG.arrPV[6].sNum[3].rPosition, percentBar := gUI.TiG.arrPV[6].sNum[3].rPercent)
    Frame (2,3 292x156)
        shows ModuleX2(extendButton := gUI.TiG.arrPV[6].sColumn[1].bExtend, retractButton := gUI.TiG.arrPV[6].sColumn[1].bRetract, stopButton := gUI.TiG.arrPV[6].sColumn[1].bStop, nameStr1 := gUI.TiG.arrPV[6].sNum[1].strName, posVal1 := gUI.TiG.arrPV[6].sNum[1].rPosition, percentBar1 := gUI.TiG.arrPV[6].sNum[1].rPercent, nameStr2 := gUI.TiG.arrPV[6].sNum[2].strName, posVal2 := gUI.TiG.arrPV[6].sNum[2].rPosition, percentBar2 := gUI.TiG.arrPV[6].sNum[2].rPercent)
    Frame (303,3 292x156)
        shows ModuleX2(extendButton := gUI.TiG.arrPV[6].sColumn[3].bExtend, retractButton := gUI.TiG.arrPV[6].sColumn[3].bRetract, stopButton := gUI.TiG.arrPV[6].sColumn[3].bStop, nameStr1 := gUI.TiG.arrPV[6].sNum[4].strName, posVal1 := gUI.TiG.arrPV[6].sNum[4].rPosition, percentBar1 := gUI.TiG.arrPV[6].sNum[4].rPercent, nameStr2 := gUI.TiG.arrPV[6].sNum[5].strName, posVal2 := gUI.TiG.arrPV[6].sNum[5].rPosition, percentBar2 := gUI.TiG.arrPV[6].sNum[5].rPercent)
    Frame (303,169 293x158)
        shows ModuleX1(extendButton := gUI.TiG.arrPV[6].sColumn[4].bExtend, retractButton := gUI.TiG.arrPV[6].sColumn[4].bRetract, stopButton := gUI.TiG.arrPV[6].sColumn[4].bStop, nameStr := gUI.TiG.arrPV[6].sNum[6].strName, posVal := gUI.TiG.arrPV[6].sNum[6].rPosition, percentBar := gUI.TiG.arrPV[6].sNum[6].rPercent)
    Frame (608,3 292x156)
        shows ModuleX2(extendButton := gUI.TiG.arrPV[6].sColumn[5].bExtend, retractButton := gUI.TiG.arrPV[6].sColumn[5].bRetract, stopButton := gUI.TiG.arrPV[6].sColumn[5].bStop, nameStr1 := gUI.TiG.arrPV[6].sNum[7].strName, posVal1 := gUI.TiG.arrPV[6].sNum[7].rPosition, percentBar1 := gUI.TiG.arrPV[6].sNum[7].rPercent, nameStr2 := gUI.TiG.arrPV[6].sNum[8].strName, posVal2 := gUI.TiG.arrPV[6].sNum[8].rPosition, percentBar2 := gUI.TiG.arrPV[6].sNum[8].rPercent)
    Frame (630,195 261x106)
        shows ModuleDTD(enable := gUI.TiG.arrPV[6].bPVD_enable, propPercent := gUI.TiG.arrPV[6].rPVDPercent)
END_VISUALIZATION

// Device/Application/display/OrigTi/Ceiling_Rail7
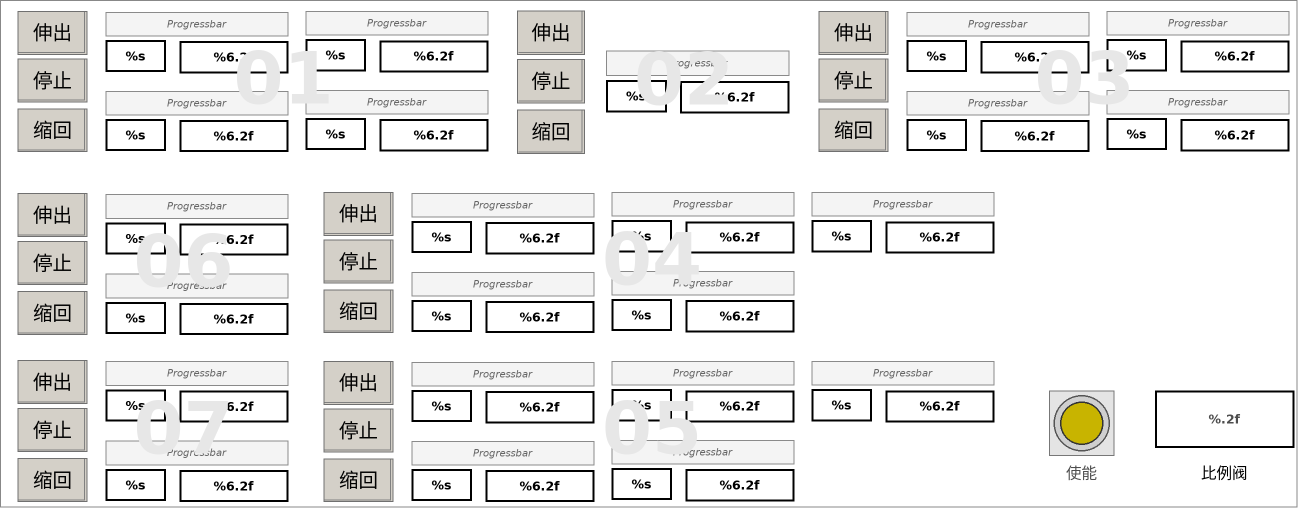
VISUALIZATION Ceiling_Rail7  // 1298x508
    Frame (0,0 492x156), "01"
        shows ModuleX4(extendButton := gUI.TiG.arrPV[7].sColumn[1].bExtend, retractButton := gUI.TiG.arrPV[7].sColumn[1].bRetract, stopButton := gUI.TiG.arrPV[7].sColumn[1].bStop, nameStr1 := gUI.TiG.arrPV[7].sNum[1].strName, posVal1 := gUI.TiG.arrPV[7].sNum[1].rPosition, percentBar1 := gUI.TiG.arrPV[7].sNum[1].rPercent, nameStr2 := gUI.TiG.arrPV[7].sNum[2].strName, posVal2 := gUI.TiG.arrPV[7].sNum[2].rPosition, percentBar2 := gUI.TiG.arrPV[7].sNum[2].rPercent, nameStr3 := gUI.TiG.arrPV[7].sNum[3].strName, posVal3 := gUI.TiG.arrPV[7].sNum[3].rPosition, percentBar3 := gUI.TiG.arrPV[7].sNum[3].rPercent, nameStr4 := gUI.TiG.arrPV[7].sNum[4].strName, posVal4 := gUI.TiG.arrPV[7].sNum[4].rPosition, percentBar4 := gUI.TiG.arrPV[7].sNum[4].rPercent)
    Frame (500,0 293x158), "02"
        shows ModuleX1(extendButton := gUI.TiG.arrPV[7].sColumn[2].bExtend, retractButton := gUI.TiG.arrPV[7].sColumn[2].bRetract, stopButton := gUI.TiG.arrPV[7].sColumn[2].bStop, nameStr := gUI.TiG.arrPV[7].sNum[5].strName, posVal := gUI.TiG.arrPV[7].sNum[5].rPosition, percentBar := gUI.TiG.arrPV[7].sNum[5].rPercent)
    Frame (801,0 492x156), "03"
        shows ModuleX4(extendButton := gUI.TiG.arrPV[7].sColumn[3].bExtend, retractButton := gUI.TiG.arrPV[7].sColumn[3].bRetract, stopButton := gUI.TiG.arrPV[7].sColumn[3].bStop, nameStr1 := gUI.TiG.arrPV[7].sNum[6].strName, posVal1 := gUI.TiG.arrPV[7].sNum[6].rPosition, percentBar1 := gUI.TiG.arrPV[7].sNum[6].rPercent, nameStr2 := gUI.TiG.arrPV[7].sNum[7].strName, posVal2 := gUI.TiG.arrPV[7].sNum[7].rPosition, percentBar2 := gUI.TiG.arrPV[7].sNum[7].rPercent, nameStr3 := gUI.TiG.arrPV[7].sNum[8].strName, posVal3 := gUI.TiG.arrPV[7].sNum[8].rPosition, percentBar3 := gUI.TiG.arrPV[7].sNum[8].rPercent, nameStr4 := gUI.TiG.arrPV[7].sNum[9].strName, posVal4 := gUI.TiG.arrPV[7].sNum[9].rPosition, percentBar4 := gUI.TiG.arrPV[7].sNum[9].rPercent)
    Frame (306,181 692x156), "04"
        shows ModuleX5(extendButton := gUI.TiG.arrPV[7].sColumn[4].bExtend, retractButton := gUI.TiG.arrPV[7].sColumn[4].bRetract, stopButton := gUI.TiG.arrPV[7].sColumn[4].bStop, nameStr1 := gUI.TiG.arrPV[7].sNum[10].strName, posVal1 := gUI.TiG.arrPV[7].sNum[10].rPosition, percentBar1 := gUI.TiG.arrPV[7].sNum[10].rPercent, nameStr2 := gUI.TiG.arrPV[7].sNum[11].strName, posVal2 := gUI.TiG.arrPV[7].sNum[11].rPosition, percentBar2 := gUI.TiG.arrPV[7].sNum[11].rPercent, nameStr3 := gUI.TiG.arrPV[7].sNum[12].strName, posVal3 := gUI.TiG.arrPV[7].sNum[12].rPosition, percentBar3 := gUI.TiG.arrPV[7].sNum[12].rPercent, nameStr4 := gUI.TiG.arrPV[7].sNum[13].strName, posVal4 := gUI.TiG.arrPV[7].sNum[13].rPosition, percentBar4 := gUI.TiG.arrPV[7].sNum[13].rPercent, nameStr5 := gUI.TiG.arrPV[7].sNum[14].strName, posVal5 := gUI.TiG.arrPV[7].sNum[14].rPosition, percentBar5 := gUI.TiG.arrPV[7].sNum[14].rPercent)
    Frame (306,350 692x156), "05"
        shows ModuleX5(extendButton := gUI.TiG.arrPV[7].sColumn[5].bExtend, retractButton := gUI.TiG.arrPV[7].sColumn[5].bRetract, stopButton := gUI.TiG.arrPV[7].sColumn[5].bStop, nameStr1 := gUI.TiG.arrPV[7].sNum[15].strName, posVal1 := gUI.TiG.arrPV[7].sNum[15].rPosition, percentBar1 := gUI.TiG.arrPV[7].sNum[15].rPercent, nameStr2 := gUI.TiG.arrPV[7].sNum[16].strName, posVal2 := gUI.TiG.arrPV[7].sNum[16].rPosition, percentBar2 := gUI.TiG.arrPV[7].sNum[16].rPercent, nameStr3 := gUI.TiG.arrPV[7].sNum[17].strName, posVal3 := gUI.TiG.arrPV[7].sNum[17].rPosition, percentBar3 := gUI.TiG.arrPV[7].sNum[17].rPercent, nameStr4 := gUI.TiG.arrPV[7].sNum[18].strName, posVal4 := gUI.TiG.arrPV[7].sNum[18].rPosition, percentBar4 := gUI.TiG.arrPV[7].sNum[18].rPercent, nameStr5 := gUI.TiG.arrPV[7].sNum[19].strName, posVal5 := gUI.TiG.arrPV[7].sNum[19].rPosition, percentBar5 := gUI.TiG.arrPV[7].sNum[19].rPercent)
    Frame (0,183 292x156), "06"
        shows ModuleX2(extendButton := gUI.TiG.arrPV[7].sColumn[6].bExtend, retractButton := gUI.TiG.arrPV[7].sColumn[6].bRetract, stopButton := gUI.TiG.arrPV[7].sColumn[6].bStop, nameStr1 := gUI.TiG.arrPV[7].sNum[20].strName, posVal1 := gUI.TiG.arrPV[7].sNum[20].rPosition, percentBar1 := gUI.TiG.arrPV[7].sNum[20].rPercent, nameStr2 := gUI.TiG.arrPV[7].sNum[21].strName, posVal2 := gUI.TiG.arrPV[7].sNum[21].rPosition, percentBar2 := gUI.TiG.arrPV[7].sNum[21].rPercent)
    Frame (0,350 292x156), "07"
        shows ModuleX2(extendButton := gUI.TiG.arrPV[7].sColumn[7].bExtend, retractButton := gUI.TiG.arrPV[7].sColumn[7].bRetract, stopButton := gUI.TiG.arrPV[7].sColumn[7].bStop, nameStr1 := gUI.TiG.arrPV[7].sNum[22].strName, posVal1 := gUI.TiG.arrPV[7].sNum[22].rPosition, percentBar1 := gUI.TiG.arrPV[7].sNum[22].rPercent, nameStr2 := gUI.TiG.arrPV[7].sNum[23].strName, posVal2 := gUI.TiG.arrPV[7].sNum[23].rPosition, percentBar2 := gUI.TiG.arrPV[7].sNum[23].rPercent)
    Frame (1035,385 261x106)
        shows ModuleDTD(enable := gUI.TiG.arrPV[7].bPVD_enable, propPercent := gUI.TiG.arrPV[7].rPVDPercent)
END_VISUALIZATION

// Device/Application/display/OrigTi/Ceiling_Rail_12
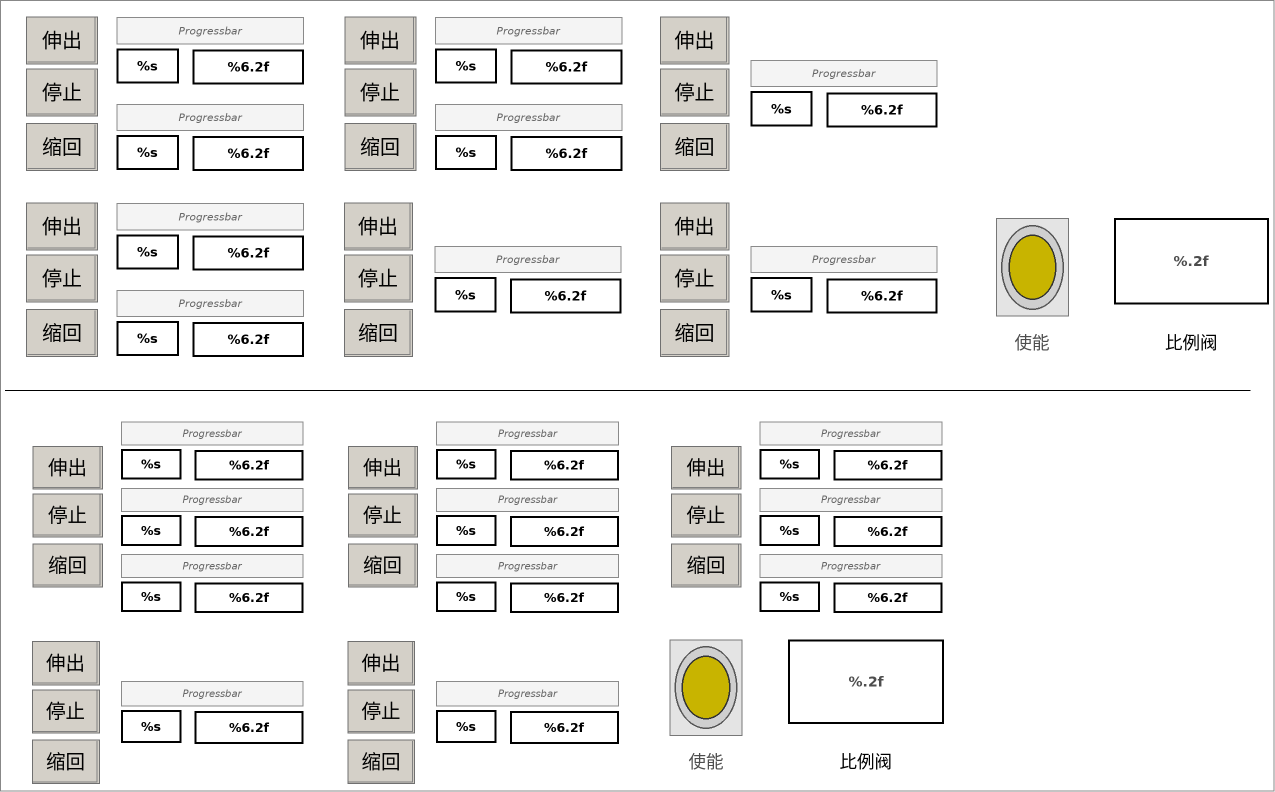
VISUALIZATION Ceiling_Rail_12  // 1275x792
    Line (5,390) (1250,390)
    Frame (3,0 1270x372)
        shows Ceiling_Rail1()
    Frame (2,403 946x387)
        shows Ceiling_Rail2()
END_VISUALIZATION

// Device/Application/display/OrigTi/Ceiling_Rail_67
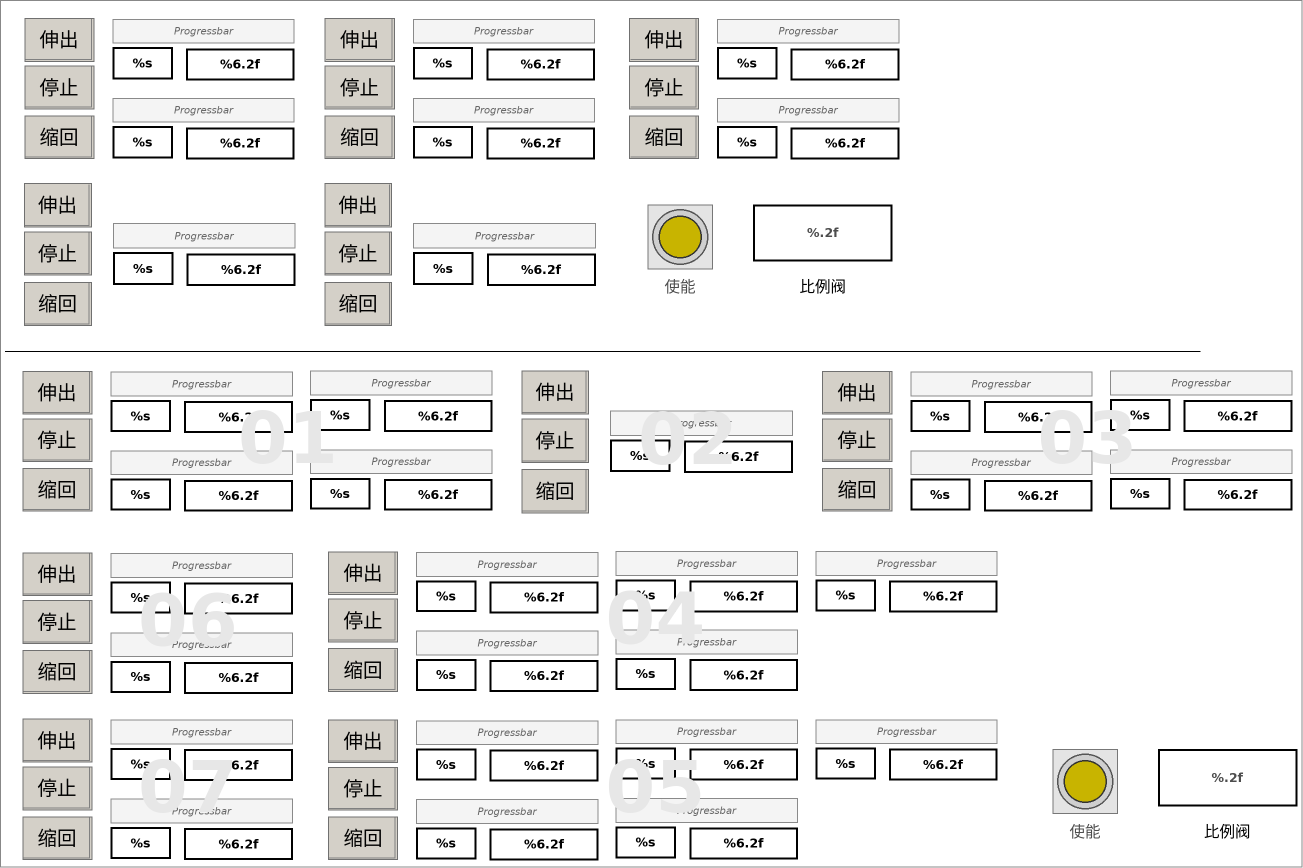
VISUALIZATION Ceiling_Rail_67  // 1303x868
    Line (5,351) (1200,351)
    Frame (5,5 900x327)
        shows Ceiling_Rail6()
    Frame (5,360 1296x506)
        shows Ceiling_Rail7()
END_VISUALIZATION

// Device/Application/display/Ceiling_Rail
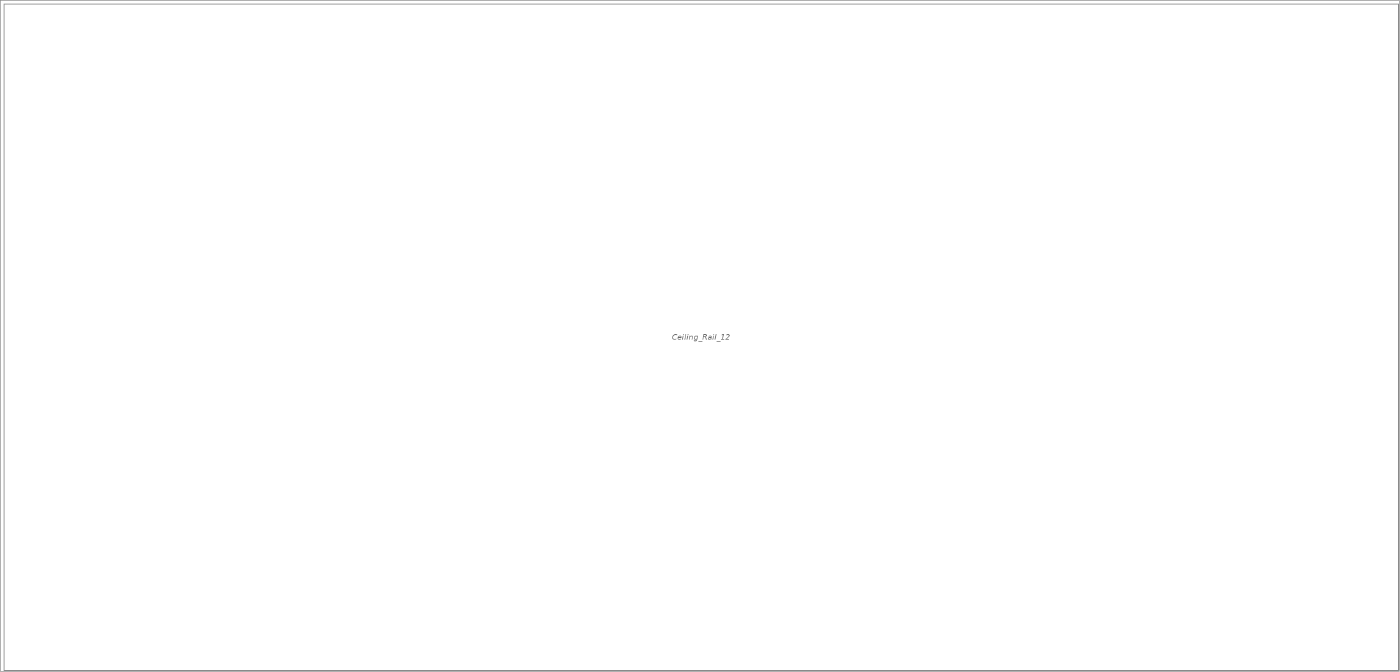
VISUALIZATION Ceiling_Rail  // 1847x887
    TabControl (5,5 1840x880)
        shows Ceiling_Rail_12()
        shows Ceiling_Rail_345()
        shows Ceiling_Rail_67()
        shows Ceiling_Rail_Plate()
        shows ManualMode()
        [0]: TabTitle=天轨1-2, ImageId=__VisualizationStyle.Element-Lamp-Lamp1-Blue-Off
        [1]: TabTitle=天轨3-5, ImageId=__VisualizationStyle.Element-Lamp-Lamp1-Blue-Off
        [2]: TabTitle=天轨6-7, ImageId=__VisualizationStyle.Element-Lamp-Lamp1-Blue-Off
        [3]: TabTitle=天轨挡板, ImageId=__VisualizationStyle.Element-Lamp-Lamp1-Blue-Off
        [4]: TabTitle=手动模式, ImageId=__VisualizationStyle.Element-Lamp-Lamp1-Blue-Off
END_VISUALIZATION

// Device/Application/display/OrigTi/Ceiling_Rail_Plate
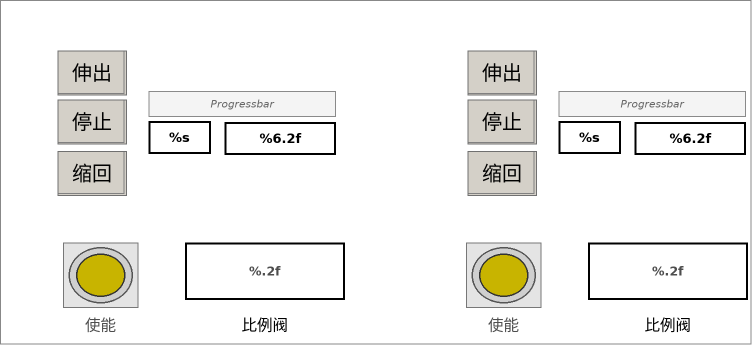
VISUALIZATION Ceiling_Rail_Plate  // 752x345
    Frame (40,40 300x160)
        shows ModuleX1(extendButton := gUI.TiG.arrPlate[1].sCmd.bExtend, retractButton := gUI.TiG.arrPlate[1].sCmd.bRetract, stopButton := gUI.TiG.arrPlate[1].sCmd.bStop, nameStr := gUI.TiG.arrPlate[1].sInfo.strName, posVal := gUI.TiG.arrPlate[1].sInfo.rPosition, percentBar := gUI.TiG.arrPlate[1].sInfo.rPercent)
    Frame (450,40 300x160)
        shows ModuleX1(extendButton := gUI.TiG.arrPlate[2].sCmd.bExtend, retractButton := gUI.TiG.arrPlate[2].sCmd.bRetract, stopButton := gUI.TiG.arrPlate[2].sCmd.bStop, nameStr := gUI.TiG.arrPlate[2].sInfo.strName, posVal := gUI.TiG.arrPlate[2].sInfo.rPosition, percentBar := gUI.TiG.arrPlate[2].sInfo.rPercent)
    Frame (47,237 300x106)
        shows ModuleDTD(enable := gUI.TiG.arrPV[6].bPVD_enable, propPercent := gUI.TiG.arrPV[6].rPVDPercent)
    Frame (450,237 300x106)
        shows ModuleDTD(enable := gUI.TiG.arrPV[1].bPVD_enable, propPercent := gUI.TiG.arrPV[1].rPVDPercent)
END_VISUALIZATION

// Device/Application/display/OrigTi/ManualMode
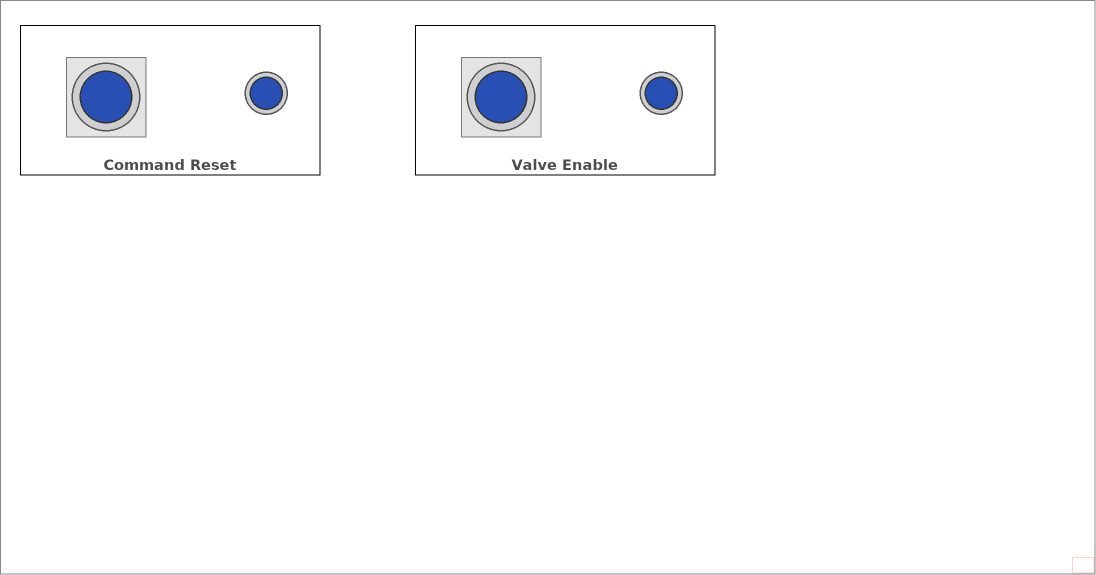
VISUALIZATION ManualMode  // 1096x575
    Rectangle (20,25 300x150), "Command Reset"
    Lamp1 (241,68 50x50), variable: gUI.sManualMode.bCmdReset, style: Lamp-Lamp1-Blue
    PushSwitchLed (66,57 80x80), variable: gUI.sManualMode.bCmdReset, behaviour: TOGGLE, style: Switch-PushSwitchLed-Blue
    Rectangle (415,25 300x150), "Valve Enable"
    Lamp1 (636,68 50x50), variable: gUI.sManualMode.bDteEnable, style: Lamp-Lamp1-Blue
    PushSwitchLed (461,57 80x80), variable: gUI.sManualMode.bDteEnable, behaviour: TOGGLE, style: Switch-PushSwitchLed-Blue
    Rectangle (1072,557 22x16)
END_VISUALIZATION
